TYPE ST_SCANNER_Statistics :
STRUCT
	nTotalReads			: UDINT;
	nValidCodes			: UDINT;
	nInvalidCodes			: UDINT;
	nDuplicateCodes		: UDINT;
	nNoCodeFound		: UDINT;
END_STRUCT
END_TYPE

(* stored: Version 1.1.0.1, ProductVersion 3.1.4024.15
   DUT ST_SCANNER_Statistics: Id {868d921b-1734-4d62-8874-b031a7e16475} *)
